// TIA Portal V19 export
DATA_BLOCK "_IOL_VM_Burk_8691r2Param"   // DB501
TITLE = Valve Monitoring Params for Burkett 8691 rev.2
{ S7_Optimized_Access := 'TRUE' }
// stored: AutoNumber false, MemoryReserve 0
   VAR RETAIN
      VM_IOL_Params : "_ILO_VM_Burkett8691rev2";
   END_VAR
BEGIN
END_DATA_BLOCK
